TYPE "OOAx_Ctrl"
VERSION : 0.1
// Block: OOAx_Ctrl
   STRUCT
      SafeStop : Bool;
      Rst : Bool;
      Homing : Bool;
      MovePlus : Bool;
      MoveMinus : Bool;
      MoveAbsolute : Bool;
      HomeMode : Int;
      HomePosition : LReal;
      MoveAbsTarget : LReal;
   END_STRUCT;

END_TYPE
